// SIMATIC S7-200 project (STEP 7-Micro/WIN), CPU 226 CN REL 02.01

ORGANIZATION_BLOCK 主程序:OB1
TITLE=
BEGIN
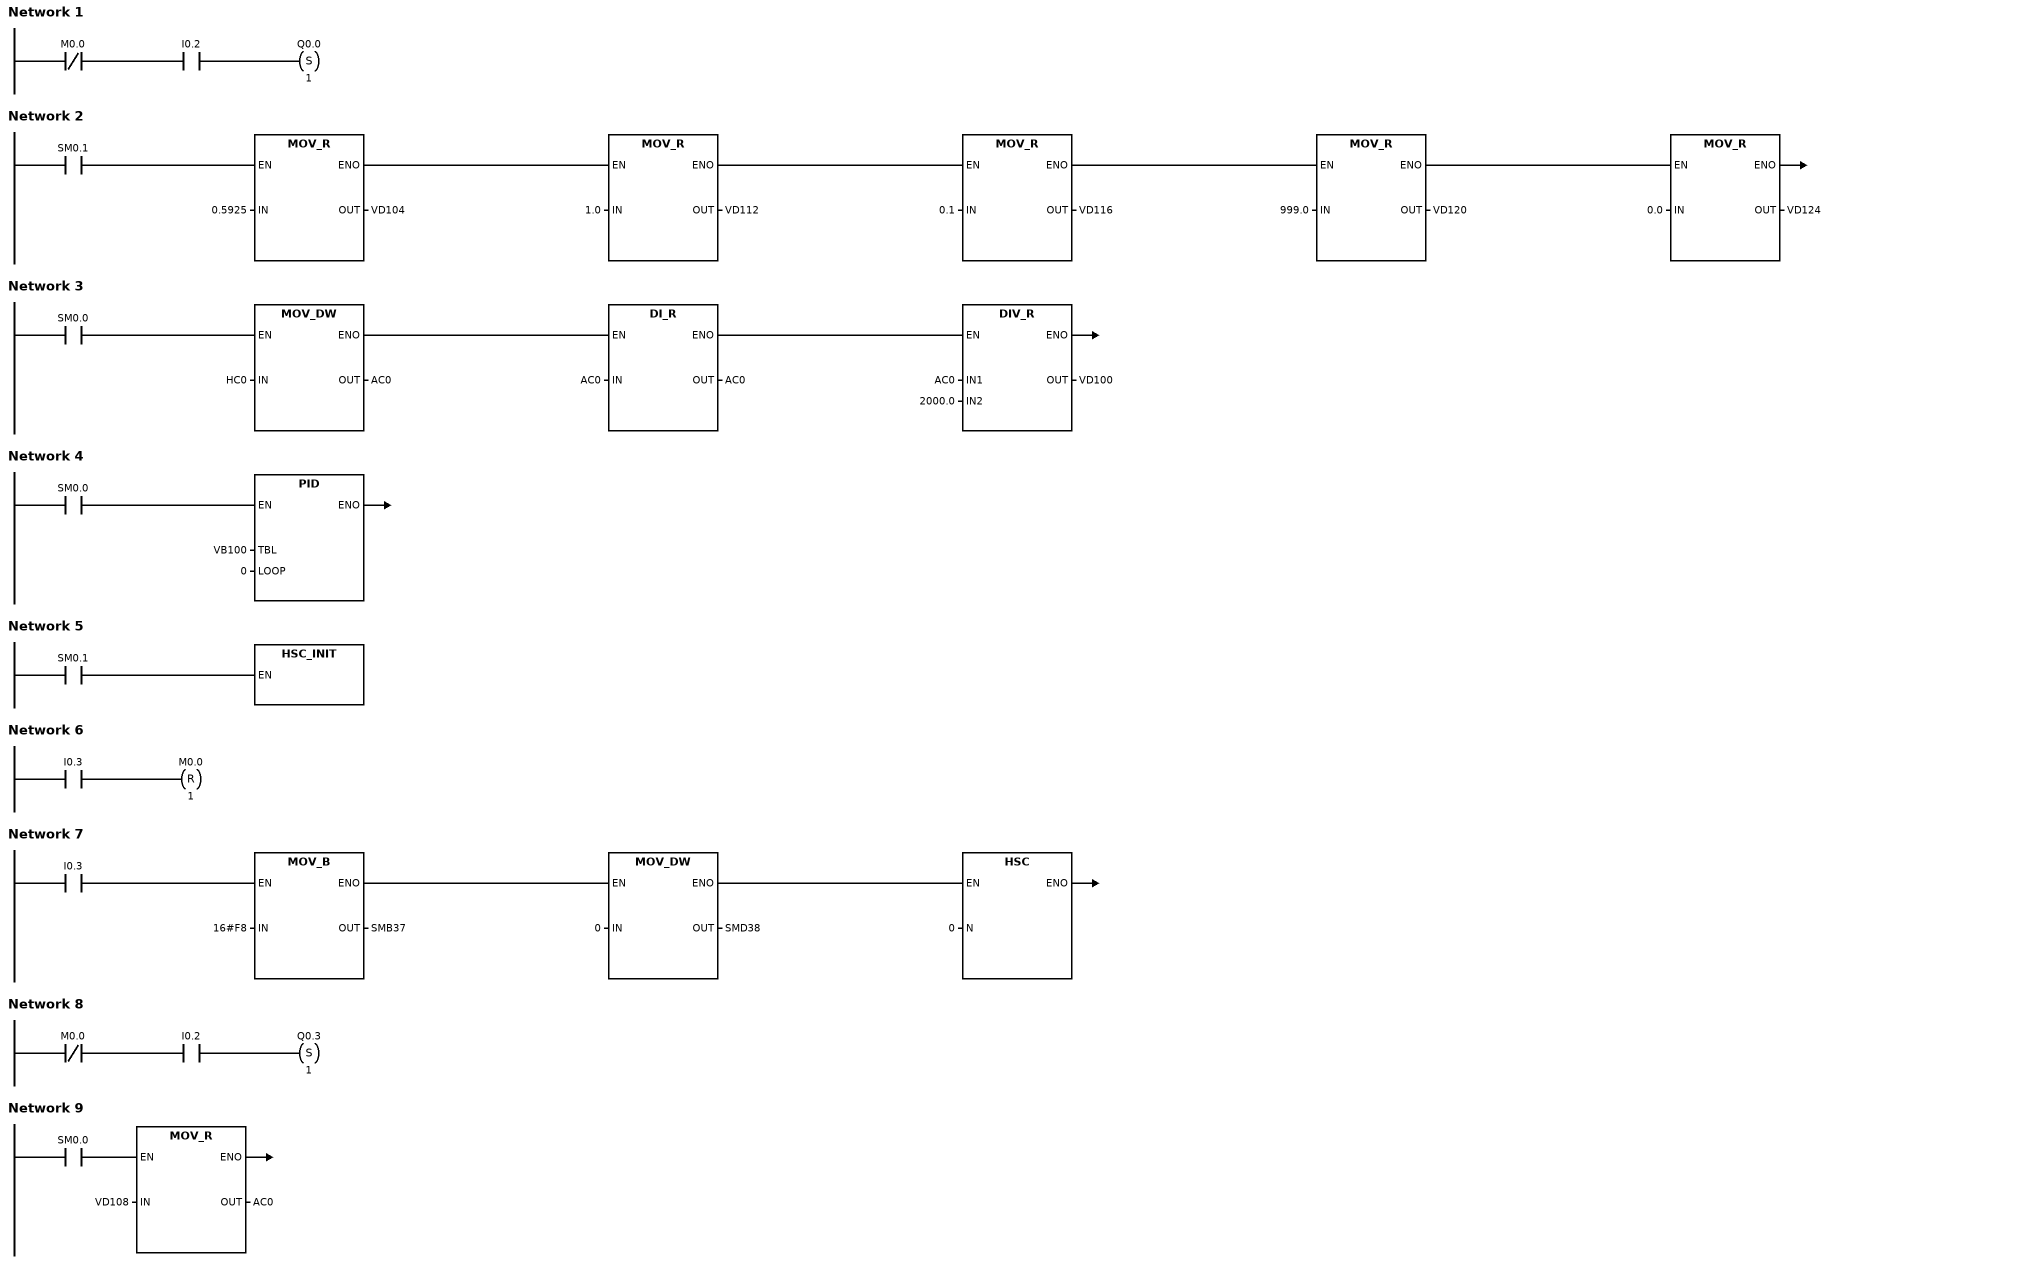
Network 1
LDN    M0.0
A      I0.2
S      Q0.0, 1
Network 2
// (network saved uncompiled; LAD cells follow)
// row 0: c0 -| |- SM0.1  c1 --  c2 [MOV_R EN:=power@row0, IN:=0.5925, ENO=>power, OUT=>VD104]  c3 --  c4 --  c5 [MOV_R EN:=power@row0, IN:=1.0, ENO=>power, OUT=>VD112]  c6 --  c7 --  c8 [MOV_R EN:=power@row0, IN:=0.1, ENO=>power, OUT=>VD116]  c9 --  c10 --  c11 [MOV_R EN:=power@row0, IN:=999.0, ENO=>power, OUT=>VD120]  c12 --  c13 --  c14 [MOV_R EN:=power@row0, IN:=0.0, ENO=>power, OUT=>VD124]  c15 ->
// row 1: c2 [box]  c5 [box]  c8 [box]  c11 [box]  c14 [box]
Network 3
// (network saved uncompiled; LAD cells follow)
// row 0: c0 -| |- SM0.0  c1 --  c2 [MOV_DW EN:=power@row0, IN:=HC0, ENO=>power, OUT=>AC0]  c3 --  c4 --  c5 [DI_R EN:=power@row0, IN:=AC0, ENO=>power, OUT=>AC0]  c6 --  c7 --  c8 [DIV_R EN:=power@row0, IN1:=AC0, IN2:=2000.0, ENO=>power, OUT=>VD100]  c9 ->
// row 1: c2 [box]  c5 [box]  c8 [box]
Network 4
LD     SM0.0
PID    VB100, 0
Network 5
LD     SM0.1
CALL   HSC_INIT:SBR2
Network 6
LD     I0.3
R      M0.0, 1
Network 7
// (network saved uncompiled; LAD cells follow)
// row 0: c0 -| |- I0.3  c1 --  c2 [MOV_B EN:=power@row0, IN:=16#F8, ENO=>power, OUT=>SMB37]  c3 --  c4 --  c5 [MOV_DW EN:=power@row0, IN:=0, ENO=>power, OUT=>SMD38]  c6 --  c7 --  c8 [HSC EN:=power@row0, N:=0, ENO=>power]  c9 ->
// row 1: c2 [box]  c5 [box]  c8 [box]
Network 8
LDN    M0.0
A      I0.2
S      Q0.3, 1
Network 9
// (network saved uncompiled; LAD cells follow)
// row 0: c0 -| |- SM0.0  c1 [MOV_R EN:=power@row0, IN:=VD108, ENO=>power, OUT=>AC0]  c2 ->
// row 1: c1 [box]
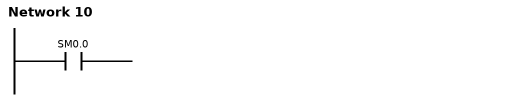
Network 10
// (network saved uncompiled; LAD cells follow)
// row 0: c0 -| |- SM0.0
END_ORGANIZATION_BLOCK

// SBR1: protected block, not included

SUBROUTINE_BLOCK HSC_INIT:SBR2
TITLE=
BEGIN
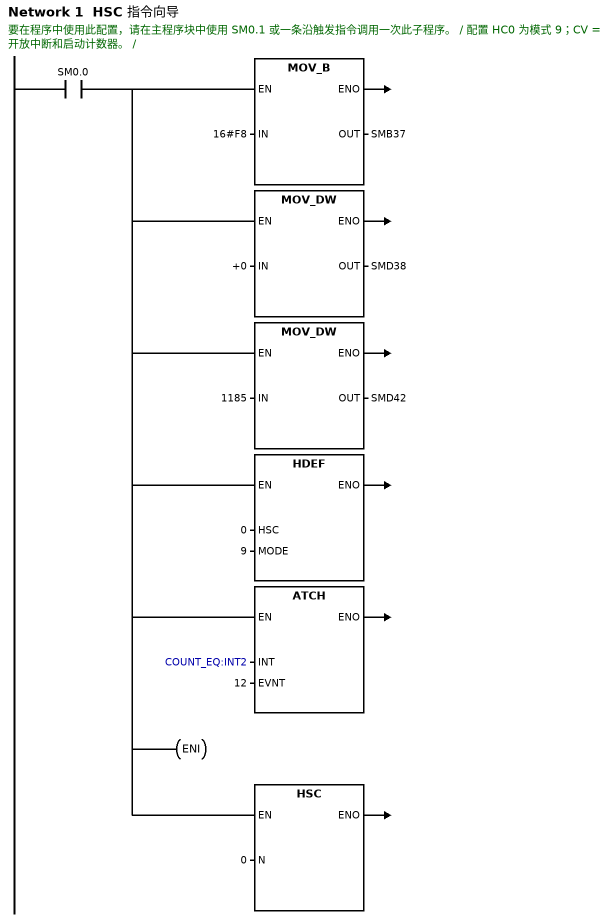
Network 1 // HSC 指令向导
// 要在程序中使用此配置，请在主程序块中使用 SM0.1 或一条沿触发指令调用一次此子程序。
// 配置 HC0 为模式 9；CV = 0； PV = 12000；增计数；
// 连接中断程序 COUNT_EQ 到事件 12 (HC0 的 CV = PV)。
// 开放中断和启动计数器。
// 
//设置控制位：增计数；4X 速率；已使能；
//装载 CV
//装载 PV
//中断程序 COUNT_EQ：HC0 的 CV = PV
// (network saved uncompiled; LAD cells follow)
// row 0: c0 -| |- SM0.0 v  c1 --  c2 [MOV_B EN:=power@row0, IN:=16#F8, ENO=>power, OUT=>SMB37]  c3 ->
// row 1: c0 ^v  c2 [box]
// row 2: c0 ^v  c1 --  c2 [MOV_DW EN:=power@row2, IN:=+0, ENO=>power, OUT=>SMD38]  c3 ->
// row 3: c0 ^v  c2 [box]
// row 4: c0 ^v  c1 --  c2 [MOV_DW EN:=power@row4, IN:=1185, ENO=>power, OUT=>SMD42]  c3 ->
// row 5: c0 ^v  c2 [box]
// row 6: c0 ^v  c1 --  c2 [HDEF EN:=power@row6, HSC:=0, MODE:=9, ENO=>power]  c3 ->
// row 7: c0 ^v  c2 [box]
// row 8: c0 ^v  c1 --  c2 [ATCH EN:=power@row8, INT:=COUNT_EQ:INT2, EVNT:=12, ENO=>power]  c3 ->
// row 9: c0 ^v  c2 [box]
// row 10: c0 ^v  c1 -(ENI)
// row 11: c0 ^  c1 --  c2 [HSC EN:=power@row11, N:=0, ENO=>power]  c3 ->
// row 12: c2 [box]
END_SUBROUTINE_BLOCK

INTERRUPT_BLOCK INT_0:INT0
TITLE=中断程序注释
BEGIN
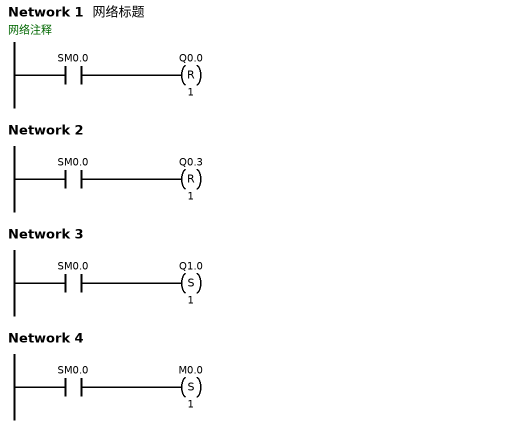
Network 1 // 网络标题
// 网络注释
LD     SM0.0
R      Q0.0, 1
Network 2
LD     SM0.0
R      Q0.3, 1
Network 3
LD     SM0.0
S      Q1.0, 1
Network 4
LD     SM0.0
S      M0.0, 1
END_INTERRUPT_BLOCK

// INT1: protected block, not included

// (further data pages could not be read)
